// TwinCAT 3 PLC project Quality_AnalyserPLC
// ProgramVersion: 3.1.4024.0
// libraries:
//   Tc2_Standard, * (Beckhoff Automation GmbH)
//   Tc2_System, * (Beckhoff Automation GmbH)
//   Tc3_Module, * (Beckhoff Automation GmbH)
// project tree:
//   DUTs/ ST_MinMax.TcDUT, ST_ProductStats.TcDUT
//   / PlcTask.TcTTO
//   POUs/ F_AnalyzeBatch.TcPOU (not stored), F_CalculateAverage.TcPOU (not stored), F_CountDefects.TcPOU (not stored), F_FindMinMax.TcPOU (not stored), MAIN.TcPOU (not stored)
// real-time tasks:
//   TASK PlcTask: cycle T#10ms, priority 20, ADS port 350

CONFIGURATION Quality_AnalyserPLC
    RESOURCE PLC ON TwinCAT3
        TASK PlcTask(INTERVAL := T#10ms, PRIORITY := 20);
        PROGRAM MAIN WITH PlcTask : MAIN;
    END_RESOURCE
END_CONFIGURATION

// ---- DUTs/ST_MinMax.TcDUT
TYPE ST_MinMax :
STRUCT
	mini : REAL;
	maxi : REAL;
END_STRUCT
END_TYPE

// ---- DUTs/ST_ProductStats.TcDUT
TYPE ST_ProductStats :
STRUCT
	averageWeight :REAL;
	minWeight : REAL;
	maxWeight : REAL;
	defectiveCount : INT;
END_STRUCT
END_TYPE
